Omron CX-Programmer project NewProject (CX-Programmer 9.50)

# PLC Mesin_Cuci_Otomatis: CP1L M

## Global symbols (name address type ; comment)
0.00 BOOL  ; START
0.01 BOOL  ; STOP
0.02 BOOL  ; SENSOR
100.01 BOOL  ; CONVEYOR
100.02 BOOL  ; BRUSH
1.00 BOOL  ; SPRAY
6.00 BOOL  ; IR

## Program NewProgram1 (cyclic task 0)

### Section Section1

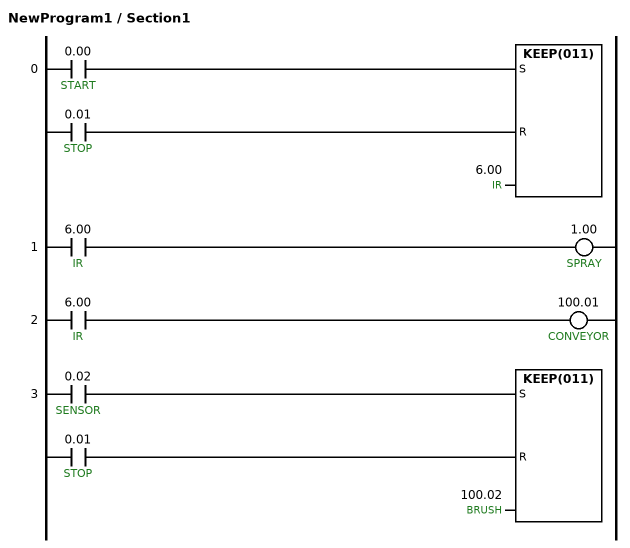
; rung 0
LD 0.00  ; START
LD 0.01  ; STOP
KEEP(011) 6.00  ; IR
; rung 1
LD 6.00  ; IR
OUT 1.00  ; SPRAY
; rung 2
LD 6.00  ; IR
OUT 100.01  ; CONVEYOR
; rung 3
LD 0.02  ; SENSOR
LD 0.01  ; STOP
KEEP(011) 100.02  ; BRUSH

### Section END
; rung 0
END(001)